(* PLC project cp_cab, Dassault Systèmes ControlBuild 2024x *)
(* stored: creationDateTime 2023-10-03T11:13:51-01:00 *)

FUNCTION_BLOCK tni_train.cp_cab
  VAR_INPUT
    keyCabEnabled : BOOL := false;
    keyCabDisabled : BOOL := false;
    rightServiceSide : BOOL := false;
    leftServiceSide : BOOL := false;
    pbDoorClosing : BOOL := false;
    speed : REAL := 0.0;
    keyCabEnabled2 : BOOL := false;
    keyCabDisabled2 : BOOL := false;
  END_VAR
  VAR_OUTPUT
    enableOpeningRightC1 : BOOL := false;
    enableOpeningLeftC1 : BOOL := false;
    enableClosingRightC1 : BOOL := false;
    enableClosingLeftC1 : BOOL := false;
  END_VAR
  VAR_OUTPUT
    cabEnabled : BOOL := false;
    cabDisabled : BOOL := false;
    cabIncoherence : BOOL := false;
  END_VAR
  VAR CONSTANT
    limitLowSpeed : REAL := 6.0;
  END_VAR

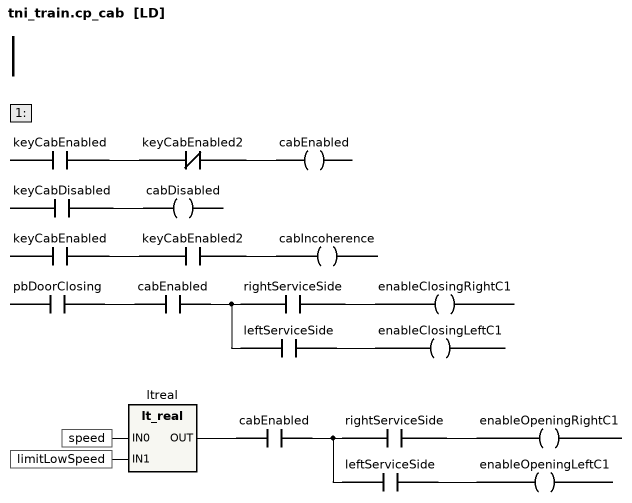
(* LD diagram, written out as Structured Text *)
1:
cabEnabled := keyCabEnabled AND NOT keyCabEnabled2;
cabDisabled := keyCabDisabled;
cabIncoherence := keyCabEnabled AND keyCabEnabled2;
ltreal(IN0 := speed, IN1 := limitLowSpeed);
enableOpeningRightC1 := ltreal.OUT AND cabEnabled AND rightServiceSide;
enableOpeningLeftC1 := ltreal.OUT AND cabEnabled AND leftServiceSide;
enableClosingRightC1 := pbDoorClosing AND cabEnabled AND rightServiceSide;
enableClosingLeftC1 := pbDoorClosing AND cabEnabled AND leftServiceSide;
END_FUNCTION_BLOCK
